// TIA Portal V21 export
DATA_BLOCK "Data_block_11"   // DB2
{ S7_Optimized_Access := 'TRUE' }
// stored: MemoryReserve 100
   VAR
      var1 : Bool;
   END_VAR
BEGIN
END_DATA_BLOCK
